// TIA Portal project "2022.06.05_计数器2" (V17)

(* hardware
DEVICE "S7-1200 station_1"  S7-1200 Station
   slot 0: "Rack_0"  S7-1200 Rack  Rack  V1.0
   slot 1: "PLC_1"  CPU 1212C DC/DC/DC  6ES7 212-1AE40-0XB0  V4.5
*)

// ===== PLC "PLC_1"  CPU 1212C DC/DC/DC =====

VAR_GLOBAL   // PLC tag table "默认变量表"
   "Tag_1" AT %I0.0 : Bool;
   "自动复位" AT %M0.0 : Bool;
   "Tag_3" AT %I0.2 : Bool;
   "Tag_4" AT %MW10 : Int;
   "Tag_5" AT %Q0.0 : Bool;
   "手动复位" AT %I0.1 : Bool;
   "初始位" AT %M1.0 : Bool;
   "Tag_2" AT %M0.1 : Bool;
   "赋值" AT %I0.3 : Bool;
   "Tag_7" AT %I0.4 : Bool;
   "加" AT %I0.5 : Bool;
   "Tag_9" AT %M10.0 : Bool;
   "减" AT %I0.6 : Bool;
   "手动复位(1)" AT %I0.7 : Bool;
   "Tag_12" AT %M10.1 : Bool;
   "当前值" AT %MW20 : Int;
   "Tag_6" AT %M0.2 : Bool;
   "5次" AT %M0.3 : Bool;
END_VAR

// folder: System blocks/Program resources

DATA_BLOCK "IEC_Counter_0_DB"   // DB1
{ S7_Optimized_Access := 'TRUE' }
AUTHOR : Simatic
FAMILY : IEC
NAME : CNTR
VERSION : 1.0
// stored: InstanceOfName IEC_COUNTER
"IEC_COUNTER"
BEGIN
END_DATA_BLOCK

DATA_BLOCK "IEC_Counter_0_DB_1"   // DB2
{ S7_Optimized_Access := 'TRUE' }
AUTHOR : Simatic
FAMILY : IEC
NAME : CNTR
VERSION : 1.0
// stored: InstanceOfName IEC_COUNTER
"IEC_COUNTER"
BEGIN
END_DATA_BLOCK

DATA_BLOCK "IEC_Counter_0_DB_2"   // DB3
{ S7_Optimized_Access := 'TRUE' }
AUTHOR : Simatic
FAMILY : IEC
NAME : CNTR
VERSION : 1.0
// stored: InstanceOfName IEC_COUNTER
"IEC_COUNTER"
BEGIN
END_DATA_BLOCK

DATA_BLOCK "IEC_Timer_0_DB"   // DB4
{ S7_Optimized_Access := 'TRUE' }
AUTHOR : Simatic
FAMILY : IEC
NAME : IEC_TMR
VERSION : 1.0
// stored: InstanceOfName IEC_TIMER
"IEC_TIMER"
BEGIN
END_DATA_BLOCK

DATA_BLOCK "IEC_Counter_0_DB_3"   // DB5
{ S7_Optimized_Access := 'TRUE' }
AUTHOR : Simatic
FAMILY : IEC
NAME : CNTR
VERSION : 1.0
// stored: InstanceOfName IEC_COUNTER
"IEC_COUNTER"
BEGIN
END_DATA_BLOCK

// folder: (top level)

ORGANIZATION_BLOCK "Main"   // OB1, LAD, ProgramCycle
TITLE = "Main Program Sweep (Cycle)"
{ S7_Optimized_Access := 'TRUE' }
VERSION : 0.1
// 启动：q0.0闪烁5次。停止（亮0.5，灭0.5）
   VAR_INPUT
      Initial_Call : Bool;   // Initial call of this OB
      Remanence : Bool;   // =True, if remanent data are available
   END_VAR
BEGIN

REGION Network 1
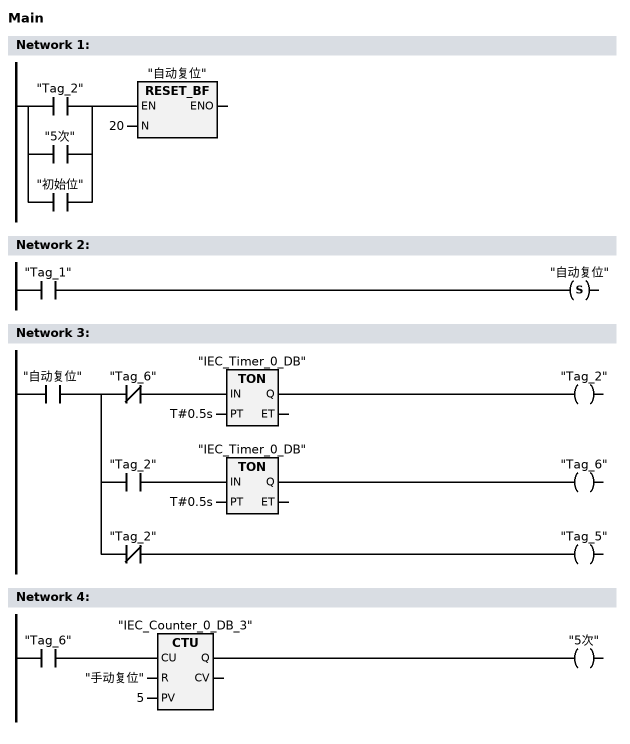
   // no SCL statement known for RBitfield: written as a call
   IF "Tag_2" OR "5次" OR "初始位" THEN RESET_BF(operand := "自动复位", n := 20); END_IF;
END_REGION

REGION Network 2
   RUNG wire#powerrail
      Contact( "Tag_1" )
      S_Coil( "自动复位" )
   END_RUNG
   // the same network as SCL:
   IF "Tag_1" THEN "自动复位" := TRUE; END_IF;
END_REGION

REGION Network 3
   "IEC_Timer_0_DB".TON(IN := "自动复位" AND NOT "Tag_6", PT := T#0.5s);
   "Tag_2" := "IEC_Timer_0_DB".Q;
   "IEC_Timer_0_DB".TON(IN := "自动复位" AND "Tag_2", PT := T#0.5s);
   "Tag_6" := "IEC_Timer_0_DB".Q;
   "Tag_5" := "自动复位" AND NOT "Tag_2";
END_REGION

REGION Network 4
   "IEC_Counter_0_DB_3".CTU(CU := "Tag_6", R := "手动复位", PV := 5);
   "5次" := "IEC_Counter_0_DB_3".Q;
END_REGION
END_ORGANIZATION_BLOCK